FUNCTION "LnkJ_Hello" : Void
{ S7_Optimized_Access := 'TRUE' }
VERSION : 0.1
   VAR_INPUT
      Seq : UInt;   // 엔벨로프 seq (1..65535, 0 = 없음)
   END_VAR

   VAR_IN_OUT
      Buf : Array[*] of Byte;   // 출력 버퍼
      Pos : DInt;   // 다음 쓸 절대 인덱스 (< 0 = 오류 유지)
      Val : "LNK_Hello";   // data
   END_VAR


BEGIN
	// GENERATED by gr-contract gen-link from message "Hello" (id 1, "LNK_Hello" sig 16#BFAD9982) - do not edit
	// {"type":"Hello","seq":<Seq>,"sig":3215825282,"data":<Val>}
	"Json_WRaw"(Buf := #Buf, Pos := #Pos, Lit := '{"type":"Hello","seq":');
	"Json_WUInt"(Buf := #Buf, Pos := #Pos, Val := #Seq);
	"Json_WRaw"(Buf := #Buf, Pos := #Pos, Lit := ',"sig":3215825282,"data":');
	"JsonW_LNK_Hello"(Buf := #Buf, Pos := #Pos, Val := #Val);
	"Json_WRaw"(Buf := #Buf, Pos := #Pos, Lit := '}');
END_FUNCTION
